{attribute 'linkalways'} 
INTERFACE I_PromiseContext

METHOD PUBLIC Reject
VAR_INPUT
	Reason : T_MAXSTRING;
END_VAR
END_METHOD

METHOD PUBLIC Resolve
VAR_INPUT
END_VAR
END_METHOD

METHOD PUBLIC ResolveWith
VAR_INPUT
	Value : ANY;
END_VAR
END_METHOD

METHOD PUBLIC TryGetEntity : BOOL
VAR_INPUT
	Key : T_MAXSTRING;
	Destination	: ANY;
END_VAR
END_METHOD

METHOD PUBLIC TryGetEntityTo : BOOL
VAR_INPUT
	Key : T_MAXSTRING;
	DestinationAddress : PVOID;
	DestinationSize : UDINT;
END_VAR
END_METHOD

METHOD PUBLIC TrySetEntity : BOOL
VAR_INPUT
	Key : T_MAXSTRING;
	Value : ANY;
END_VAR
END_METHOD

END_INTERFACE

(* stored: Version 1.1.0.1, ProductVersion 3.1.4024.12
   Itf I_PromiseContext: Id {ac6c8482-60f6-4d24-803f-071e8ab643bb}
   Method Reject: Id {0b79950d-7e9e-41f6-a877-3005abe5e686}
   Method Resolve: Id {0ddc6a64-376f-4da1-b1fc-4ee93fa62f61}
   Method ResolveWith: Id {565da8d7-902a-4c61-9c04-96db233562a2}
   Method TryGetEntity: Id {d468ed09-b31e-4279-af65-3e47e517028a}
   Method TryGetEntityTo: Id {bdf8d47b-dd1a-44ff-b6e1-ca362b20f84c}
   Method TrySetEntity: Id {7edba61f-afac-4a0d-acfc-d6dbf60d35c2} *)
